PROGRAM P_Demo_FB_HVACCirculationPump
VAR
    fb : FB_HVACCirculationPump;                            // 被演示 FB 实例
    eDataSecurityType_in : E_HVACDataSecurityType ;
    bSetDefault_in : BOOL := FALSE;
    bEnable_in : BOOL := FALSE;
    bAuto_in : BOOL := FALSE;
    eCtrlModeActuator_in : E_HVACActuatorMode ;
    rOutsideTemp_in : REAL := 0.0;
    rValvePosition_in : REAL := 0.0;
    bFeedbPump_in : BOOL := FALSE;
    bPumpProtec_in : BOOL := FALSE;
    bAntiBlocking_in : BOOL := FALSE;
    bManSwitch_in : BOOL := FALSE;
    bCtrlVoltage_in : BOOL := FALSE;
    bReset_in : BOOL := FALSE;
    tStopDelay_io : TIME := T#0S;
    tFeedbPumpDelay_io : TIME := T#0S;
    rOutsideTempLimit_io : REAL := 0.0;
    rValvePositionLimit_io : REAL := 0.0;
    eReqOutsideTemp_io : E_HVACReqOutsideTemp ;
    eReqValve_io : E_HVACReqValve ;
    bPump_out : BOOL;
    byState_out : BYTE;
    bStateManSwitch_out : BOOL;
    bReqOutsideTemp_out : BOOL;
    bReqValve_out : BOOL;
    eStateModeActuator_out : E_HVACActuatorMode;
    bErrorPumpProtec_out : BOOL;
    bErrorPumpFeedb_out : BOOL;
    bErrorGeneral_out : BOOL;
    byError_out : BYTE;
    bInvalidParameter_out : BOOL;
END_VAR

// ============================================================================
// Tc2_HVAC.FB_HVACCirculationPump 演示程序
// ============================================================================
// 场景：把本 FB 实例化到一个 PLC 程序里，每周期单次调用；按需要把 VAR_INPUT 与
//       VAR_IN_OUT 接到工程信号；VAR_OUTPUT 写入对应监视变量。
// 价值：使用本 FB 比手写状态机 / 控制算法节省大量代码；与 Tc2_HVAC 体系内其它 FB
//       直接对接，命名 / 持久化 / 模式仲裁等约定一致。具体语义见 FB_HVACCirculationPump.md 主文档。
// 验证步骤：
//   1. 右键 PLC 项目下 POUs 文件夹 → Add → Existing Item → 选本 .TcPOU 文件
//   2. 引用 Tc2_HVAC（References → Add library）
//   3. 编译 → 登录 → 运行
//   4. 在线写各 *_in 输入信号触发 FB；在线 monitor *_out 引脚观察状态
// ============================================================================

fb(
    eDataSecurityType := eDataSecurityType_in,
    bSetDefault := bSetDefault_in,
    bEnable := bEnable_in,
    bAuto := bAuto_in,
    eCtrlModeActuator := eCtrlModeActuator_in,
    rOutsideTemp := rOutsideTemp_in,
    rValvePosition := rValvePosition_in,
    bFeedbPump := bFeedbPump_in,
    bPumpProtec := bPumpProtec_in,
    bAntiBlocking := bAntiBlocking_in,
    bManSwitch := bManSwitch_in,
    bCtrlVoltage := bCtrlVoltage_in,
    bReset := bReset_in,
    tStopDelay := tStopDelay_io,
    tFeedbPumpDelay := tFeedbPumpDelay_io,
    rOutsideTempLimit := rOutsideTempLimit_io,
    rValvePositionLimit := rValvePositionLimit_io,
    eReqOutsideTemp := eReqOutsideTemp_io,
    eReqValve := eReqValve_io,
    bPump => bPump_out,
    byState => byState_out,
    bStateManSwitch => bStateManSwitch_out,
    bReqOutsideTemp => bReqOutsideTemp_out,
    bReqValve => bReqValve_out,
    eStateModeActuator => eStateModeActuator_out,
    bErrorPumpProtec => bErrorPumpProtec_out,
    bErrorPumpFeedb => bErrorPumpFeedb_out,
    bErrorGeneral => bErrorGeneral_out,
    byError => byError_out,
    bInvalidParameter => bInvalidParameter_out
);

END_PROGRAM

(* stored: Version 1.1.0.1, ProductVersion 3.1.4024.5
   POU P_Demo_FB_HVACCirculationPump: Id {6d0d9d2c-c6a9-58ab-a741-4272a1387caa}, SpecialFunc None *)
